FUNCTION_BLOCK TEST_SELI (* Test SEL functions on integer types *)
  (* Standard: IEC 61499-1 *)
  (* Version 0.0, 2006-09-14, JHC, Holobloc Inc *)
  (* Compiler header: package fb.rt.test; *)
  (* Compiler classdef: SimpleFB *)
  (* Compiler Java Sun JDK 1.5.0 *)
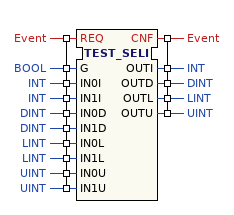
  EVENT_INPUT
    REQ WITH IN1I, IN0I, IN0D, IN1L, IN0L, IN1U, IN0U, G, IN1D;
  END_EVENT
  EVENT_OUTPUT
    CNF WITH OUTI, OUTD, OUTL, OUTU;
  END_EVENT
  VAR_INPUT
    G : BOOL; (* Selection gate *)
    IN0I : INT;
    IN1I : INT;
    IN0D : DINT;
    IN1D : DINT;
    IN0L : LINT;
    IN1L : LINT;
    IN0U : UINT;
    IN1U : UINT;
  END_VAR
  VAR_OUTPUT
    OUTI : INT;
    OUTD : DINT;
    OUTL : LINT;
    OUTU : UINT;
  END_VAR
  ALGORITHM REQ IN FBD:
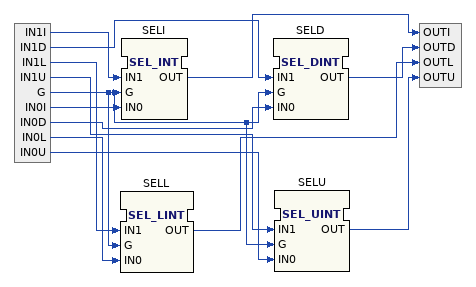
    FBS
      SELI : SEL_INT;
      SELD : SEL_DINT;
      SELL : SEL_LINT;
      SELU : SEL_UINT;
    END_FBS
    DATA_CONNECTIONS
      IN1I TO SELI.IN1;
      SELI.OUT TO OUTI;
      IN1D TO SELD.IN1;
      SELD.OUT TO OUTD;
      IN1L TO SELL.IN1;
      SELL.OUT TO OUTL;
      IN1U TO SELU.IN1;
      SELU.OUT TO OUTU;
      G TO SELI.G;
      IN0I TO SELI.IN0;
      G TO SELD.G;
      IN0D TO SELD.IN0;
      G TO SELL.G;
      IN0L TO SELL.IN0;
      G TO SELU.G;
      IN0U TO SELU.IN0;
    END_CONNECTIONS
  END_ALGORITHM
END_FUNCTION_BLOCK
